DATA_BLOCK "TRUNK3"
{ S7_Optimized_Access := 'TRUE' }
AUTHOR : RP
VERSION : 0.4
NON_RETAIN
"TRUNK-PCT"

BEGIN

END_DATA_BLOCK
